TYPE StrRampTime :
STRUCT
	rampTimeNegMaxMin	:	TIME;
	rampTimeNegMinMax	:	TIME;
	rampTimePosMaxMin	:	TIME;
	rampTimePosMinMax	:	TIME;
END_STRUCT
END_TYPE

(* stored: Version 1.1.0.1, ProductVersion 3.1.4024.12
   DUT StrRampTime: Id {dd49b41a-d94a-42ba-a56f-6003d9cdaaa8} *)
